TYPE "Positioning_EPOS_Machine_DataOut"
VERSION : 0.1
// Block: Positioning_EPOS_Machine_DataOut
   STRUCT
      Fan_M_Contactor : Bool;
   END_STRUCT;

END_TYPE
